{attribute 'linkalways'} 
{attribute 'no_explicit_call' := 'This FB is a CLASS and must be accessed using methods or properties'}
{attribute 'enable_dynamic_creation'}
FUNCTION_BLOCK FINAL LE_LINT EXTENDS Node
VAR
	in1 : _LINT(0);
	in2 : _LINT(0);
	out : _BOOL(FALSE);
END_VAR

METHOD PUBLIC Clone : I_Node
VAR
	pNode : POINTER TO LE_LINT;
END_VAR
pNode := __NEW(LE_LINT);
Clone := pNode^;
END_METHOD

METHOD FB_init : BOOL
VAR_INPUT
	bInitRetains : BOOL; // if TRUE, the retain variables are initialized (warm start / cold start)
	bInCopyCode : BOOL;  // if TRUE, the instance afterwards gets moved into the copy code (online change)
END_VAR
AddInput('in1',THIS^.in1);
AddInput('in2',THIS^.in2);
AddOutput('out', THIS^.out);
END_METHOD

METHOD PROTECTED OnExecute
VAR
END_VAR
out.Value := in1.Value <= in2.Value;
END_METHOD

END_FUNCTION_BLOCK

(* stored: Version 1.1.0.1, ProductVersion 3.1.4024.15
   POU LE_LINT: Id {23e297ef-aa9f-4633-9c88-de3271cc1d3e}, SpecialFunc None
   Folder Constructor: Id {14d8c784-b64c-47dc-bf78-3bad0165d609}
   Method Clone: Id {b4377d97-8e15-4f9a-93d8-850de734cb60}
   Method FB_init: Id {f1a36d12-6d03-4020-8d89-d28baad7e870}
   Method OnExecute: Id {8e16c29c-1f36-41d6-b5f7-815e7b1f3317} *)
